{attribute 'no_explicit_call' := 'do not call this POU directly'}
FUNCTION_BLOCK INTERNAL FB_RpcProxy IMPLEMENTS I_RpcProxy
VAR_INPUT
END_VAR
VAR_OUTPUT
END_VAR
VAR
	fbRpcSnappyVerify		: FB_RPC_Dynamic;
	sAmsNetID				: T_AmsNetID 			:= Param_TcHaxx_Snappy.cSnappyVerifyAmsNetID;
	nAmsPort				: T_AmsPort				:= Param_TcHaxx_Snappy.cSnappyVerifyPort;
	sInstancePathLocalField	: STRING				:= Param_TcHaxx_Snappy.cSnappyVerifyInstancePath;
	sSymbolLocalField		: STRING				:= Param_TcHaxx_Snappy.cSnappyVerifySymbol;
	bIsConfiguredField		: BOOL					:= FALSE;
	stVerificationResult	: ST_VerificationResult;
	itfTestFrameWorkField	: I_TestFrameWorkAdapter;
END_VAR

PROPERTY bIsConfigured : BOOL
GET
bIsConfigured := bIsConfiguredField;
END_GET
END_PROPERTY

METHOD GetVerificationResult : HRESULT
VAR_OUTPUT
	stResult : ST_VerificationResult;
END_VAR

VAR
	stAdsStatus	: TcHaxx_rplc.ST_AdsStatus;
END_VAR
GetVerificationResult := S_PENDING;

stAdsStatus := THIS^.fbRpcSnappyVerify.Invoke();

IF NOT stAdsStatus.bBusy AND NOT stAdsStatus.bError THEN
	GetVerificationResult := S_OK;
	stResult := stVerificationResult;
	RETURN;
ELSIF stAdsStatus.bError THEN
	GetVerificationResult := TO_DINT(stAdsStatus.nError);
	IF GetVerificationResult > 0 THEN
		GetVerificationResult := TO_DINT(TO_UDINT(GetVerificationResult) OR 16#98110000);
	END_IF
	RETURN;
END_IF
END_METHOD

PROPERTY itfTestFrameWorkAdapter : I_TestFrameWorkAdapter
GET
itfTestFrameWorkAdapter := THIS^.itfTestFrameWorkField;
END_GET
SET
THIS^.itfTestFrameWorkField := itfTestFrameWorkAdapter;
END_SET
END_PROPERTY

METHOD Verify : HRESULT
VAR_INPUT CONSTANT
	sToVerify			: REFERENCE TO T_VerifyContent;
END_VAR
VAR
	hr			: HRESULT;
	stAdsStatus	: TcHaxx_rplc.ST_AdsStatus;
	
	
	sTestSuiteName : STRING(Param_TcHaxx_Snappy.cSnappyVerificationTestSuiteLength) := 'ATestSuiteName';
	sTestName : STRING(Param_TcHaxx_Snappy.cSnappyVerificationTestNameLength) := 'ATestName';
END_VAR
IF NOT bIsConfiguredField THEN
	hr := fbRpcSnappyVerify.Configure()
			.WithAmsNetId(sAmsNetId:= THIS^.sAmsNetID)
			.WithAmsPort(nAmsPort:= THIS^.nAmsPort)
			.WithSymbolPath(sInstancePath:= THIS^.sInstancePathLocalField, sSymbol:= THIS^.sSymbolLocalField)
			.Build();
	bIsConfiguredField := SUCCEEDED(hr);
END_IF;

IF NOT bIsConfigured THEN
	Verify := E_HRESULTAdsErr.NOTINIT;
	RETURN;
END_IF

IF itfTestFrameWorkField <> NULL THEN
	sTestSuiteName 	:= itfTestFrameWorkField.sTestSuiteName;
	sTestName 		:= itfTestFrameWorkField.sTestName;
END_IF

stAdsStatus := fbRpcSnappyVerify.VarInput(anyArg:= sTestSuiteName)
								.VarInput(anyArg:= sTestName)
							 	.VarInput(anyArg:= sToVerify)
								.ReturnValue(anyRetVal:= stVerificationResult)
								.Invoke();
IF stAdsStatus.bError THEN
	Verify := TO_DINT(stAdsStatus.nError);
	RETURN;
END_IF

Verify := S_PENDING;
END_METHOD

END_FUNCTION_BLOCK

(* stored: Version 1.1.0.1, ProductVersion 3.1.4026.18
   POU FB_RpcProxy: Id {f9e7075c-2104-427f-9a7e-5e84f1a64890}, SpecialFunc None
   Property bIsConfigured: Id {66d99f6c-2f7b-4335-8601-3cb01d592de5}
   Get Get: Id {b1f9bb6c-7f5e-474a-9938-247984a86174}
   Method GetVerificationResult: Id {a7278404-bd08-4a34-9891-a82b07ef5350}
   Property itfTestFrameWorkAdapter: Id {6a7e0fc7-c801-46b8-b597-9bc5cb4f77dd}
   Get Get: Id {1244a42b-57f8-4833-930f-e5d7db6210d1}
   Set Set: Id {8a513147-2384-409b-9700-08b643e3efa9}
   Method Verify: Id {1f2ed438-c0f1-406f-9917-7be1f3353347} *)
